Yaskawa INFORM job: FAT.JBI

/JOB
//NAME FAT
///FOLDERNAME INNE
//POS
///NPOS 0,0,0,0,0,0
//INST
///DATE 2023/10/04 15:16
///ATTR SC,RW,RJ
////FRAME ROBOT
NOP
CALL JOB:LEAVE_CAMERA
PAUSE
CALL JOB:CLEAN-R1
PAUSE
CALL JOB:MOTOTAC1
PAUSE
CALL JOB:GET_CAMERA
PAUSE
CALL JOB:SVETS
PAUSE
CALL JOB:R1-HOME
PAUSE
CALL JOB:R1-ST1-SAFE
PAUSE
CALL JOB:R1-ST2-SAFE
PAUSE
CALL JOB:SR-ARC-1
PAUSE
CALL JOB:TSYNC-R-TEST
PAUSE
CALL JOB:SYNCS1
PAUSE
CALL JOB:S1
END
